// TwinCAT 3 PLC project InheritancePractice
// ProgramVersion: 3.1.4024.0
// libraries:
//   Tc2_Standard, * (Beckhoff Automation GmbH)
//   Tc2_System, * (Beckhoff Automation GmbH)
//   Tc3_Module, * (Beckhoff Automation GmbH)
// project tree:
//   / PlcTask.TcTTO
//   POUs/ FB_Car.TcPOU, FB_PetrolEngine.TcPOU, FB_Vehicle.TcPOU, MAIN.TcPOU
// (motion and I/O tree: see PLC project functionblockpractice)
// real-time tasks:
//   TASK PlcTask: cycle T#10ms, priority 20, ADS port 350
//   TASK PlcTask2: cycle T#10ms, priority 22, ADS port 352
//   TASK PlcTask1: cycle T#10ms, priority 21, ADS port 351
//   TASK PlcTask3: cycle T#10ms, priority 23, ADS port 353
//   TASK PlcTask4: cycle T#10ms, priority 24, ADS port 354

CONFIGURATION InheritancePractice
    RESOURCE PLC ON TwinCAT3
        TASK PlcTask(INTERVAL := T#10ms, PRIORITY := 24);
        PROGRAM MAIN WITH PlcTask : MAIN;
    END_RESOURCE
END_CONFIGURATION

// ---- POUs/MAIN.TcPOU
PROGRAM MAIN
VAR
	fbCar : FB_Car := (fFuelKilometerLimit := 4853453645);
	fbEngine : FB_PetrolEngine;
	bStart : BOOL;
	bDrive : BOOL;
END_VAR


IF bStart THEN
	fbCar.Start();
	fbCar(fbEngine := fbEngine);
END_IF

END_PROGRAM

// ---- POUs/FB_Car.TcPOU
FUNCTION_BLOCK FB_Car EXTENDS FB_Vehicle


VAR_IN_OUT
	fbEngine : FB_PetrolEngine;
END_VAR
VAR
	fCurrentFuelLimit : REAL := 42342423;
END_VAR


IF bMoving THEN
	fCurrentFuelLimit := fCurrentFuelLimit - 20;
END_IF

METHOD Feuling : BOOL
VAR_INPUT
END_VAR
bMoving := FALSE;
fCurrentFuelLimit := fFuelKilometerLimit;
END_METHOD

END_FUNCTION_BLOCK

// ---- POUs/FB_Vehicle.TcPOU
FUNCTION_BLOCK FB_Vehicle

VAR
	bRunning : BOOL;
	fFuelKilometerLimit : REAL;
	bMoving : BOOL;
END_VAR

METHOD DriveMode : BOOL
VAR_INPUT
END_VAR
IF bMoving THEN
	bMoving := FALSE;
	ELSE
	bMoving := TRUE;
END_IF
END_METHOD

METHOD Feuling : BOOL
VAR_INPUT
END_VAR
END_METHOD

METHOD Start : BOOL
VAR_INPUT
END_VAR
bRunning := TRUE;
Start := TRUE;
END_METHOD

METHOD Stop : BOOL
VAR_INPUT
END_VAR
bRunning := FALSE;
Stop :=  TRUE;
END_METHOD

END_FUNCTION_BLOCK

// ---- POUs/FB_PetrolEngine.TcPOU
FUNCTION_BLOCK FB_PetrolEngine

VAR
	nEngineCc : INT;
	fConsumption : REAL := 20;
END_VAR

END_FUNCTION_BLOCK
